// TIA Portal V18 export
// export: Created 2026-06-23T08:49:31.5753416Z, ExportSetting WithDefaults, DisplayName Totally Integrated Automation Portal, DisplayVersion V18, DisplayName TIA Portal Openness, DisplayVersion V18, DisplayName TIA Portal Version Control Interface, DisplayVersion V18, DisplayName STEP 7 Professional, DisplayVersion V18, DisplayName STEP 7 Safety, DisplayVersion V18, DisplayName WinCC Professional, DisplayVersion V18
FUNCTION "FC_Manual_Control_PLC2" : Void   // FC62, LAD
{ S7_Optimized_Access := 'TRUE' }
VERSION : 0.1
// stored: AutoNumber true, IsIECCheckEnabled false, SetENOAutomatically false, UDAEnableTagReadback false
BEGIN

REGION Network 1: Xác định trạng thái Manual Mode Active PLC2
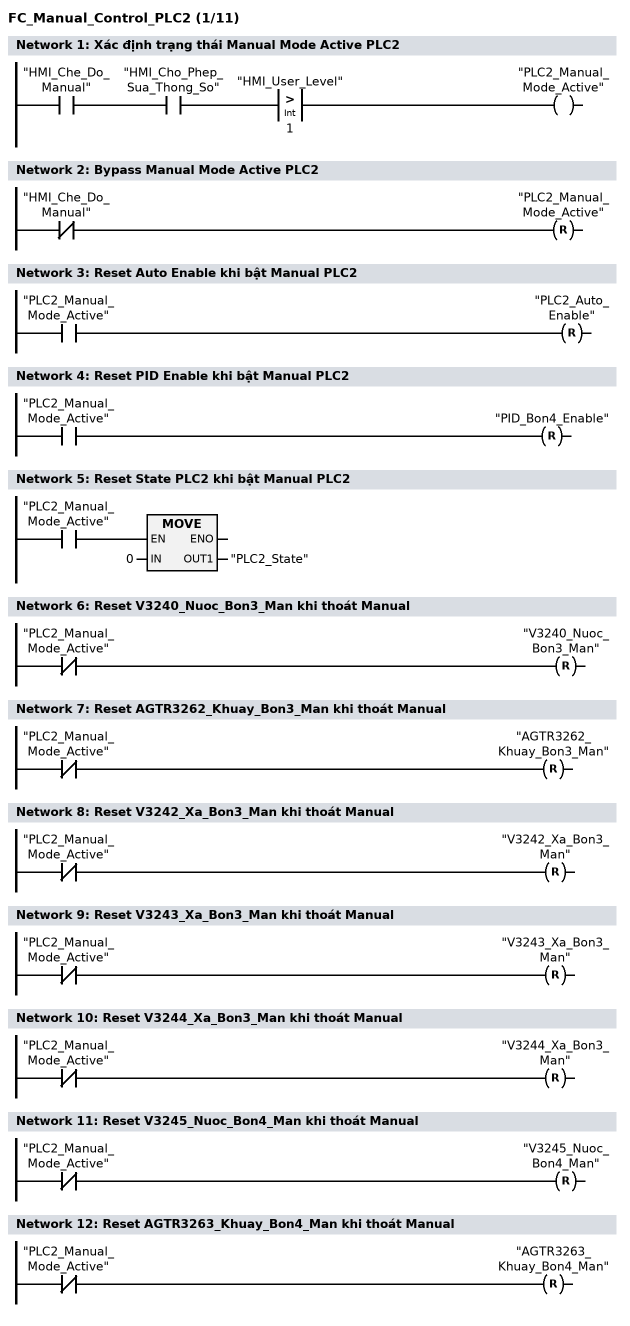
   RUNG wire#powerrail
      Contact( "HMI_Che_Do_Manual" )
      Contact( "HMI_Cho_Phep_Sua_Thong_So" )
      { S7_Templates := "SrcType := Int" } GT_Contact(in1 := "HMI_User_Level", in2 := 1)
      Coil( "PLC2_Manual_Mode_Active" )
   END_RUNG
   // the same network as SCL:
   "PLC2_Manual_Mode_Active" := "HMI_Che_Do_Manual" AND "HMI_Cho_Phep_Sua_Thong_So" AND ("HMI_User_Level" > 1);
END_REGION

REGION Network 2: Bypass Manual Mode Active PLC2
   RUNG wire#powerrail
      I_Contact( "HMI_Che_Do_Manual" )
      R_Coil( "PLC2_Manual_Mode_Active" )
   END_RUNG
   // the same network as SCL:
   IF NOT "HMI_Che_Do_Manual" THEN "PLC2_Manual_Mode_Active" := FALSE; END_IF;
END_REGION

REGION Network 3: Reset Auto Enable khi bật Manual PLC2
   RUNG wire#powerrail
      Contact( "PLC2_Manual_Mode_Active" )
      R_Coil( "PLC2_Auto_Enable" )
   END_RUNG
   // the same network as SCL:
   IF "PLC2_Manual_Mode_Active" THEN "PLC2_Auto_Enable" := FALSE; END_IF;
END_REGION

REGION Network 4: Reset PID Enable khi bật Manual PLC2
   RUNG wire#powerrail
      Contact( "PLC2_Manual_Mode_Active" )
      R_Coil( "PID_Bon4_Enable" )
   END_RUNG
   // the same network as SCL:
   IF "PLC2_Manual_Mode_Active" THEN "PID_Bon4_Enable" := FALSE; END_IF;
END_REGION

REGION Network 5: Reset State PLC2 khi bật Manual PLC2
   RUNG wire#powerrail
      Contact( "PLC2_Manual_Mode_Active" )
      { S7_GenerateENO := "TRUE" } Move(in := 0, out1 => "PLC2_State")
   END_RUNG
   // the same network as SCL:
   IF "PLC2_Manual_Mode_Active" THEN "PLC2_State" := 0; END_IF;
END_REGION

REGION Network 6: Reset V3240_Nuoc_Bon3_Man khi thoát Manual
   RUNG wire#powerrail
      I_Contact( "PLC2_Manual_Mode_Active" )
      R_Coil( "V3240_Nuoc_Bon3_Man" )
   END_RUNG
   // the same network as SCL:
   IF NOT "PLC2_Manual_Mode_Active" THEN "V3240_Nuoc_Bon3_Man" := FALSE; END_IF;
END_REGION

REGION Network 7: Reset AGTR3262_Khuay_Bon3_Man khi thoát Manual
   RUNG wire#powerrail
      I_Contact( "PLC2_Manual_Mode_Active" )
      R_Coil( "AGTR3262_Khuay_Bon3_Man" )
   END_RUNG
   // the same network as SCL:
   IF NOT "PLC2_Manual_Mode_Active" THEN "AGTR3262_Khuay_Bon3_Man" := FALSE; END_IF;
END_REGION

REGION Network 8: Reset V3242_Xa_Bon3_Man khi thoát Manual
   RUNG wire#powerrail
      I_Contact( "PLC2_Manual_Mode_Active" )
      R_Coil( "V3242_Xa_Bon3_Man" )
   END_RUNG
   // the same network as SCL:
   IF NOT "PLC2_Manual_Mode_Active" THEN "V3242_Xa_Bon3_Man" := FALSE; END_IF;
END_REGION

REGION Network 9: Reset V3243_Xa_Bon3_Man khi thoát Manual
   RUNG wire#powerrail
      I_Contact( "PLC2_Manual_Mode_Active" )
      R_Coil( "V3243_Xa_Bon3_Man" )
   END_RUNG
   // the same network as SCL:
   IF NOT "PLC2_Manual_Mode_Active" THEN "V3243_Xa_Bon3_Man" := FALSE; END_IF;
END_REGION

REGION Network 10: Reset V3244_Xa_Bon3_Man khi thoát Manual
   RUNG wire#powerrail
      I_Contact( "PLC2_Manual_Mode_Active" )
      R_Coil( "V3244_Xa_Bon3_Man" )
   END_RUNG
   // the same network as SCL:
   IF NOT "PLC2_Manual_Mode_Active" THEN "V3244_Xa_Bon3_Man" := FALSE; END_IF;
END_REGION

REGION Network 11: Reset V3245_Nuoc_Bon4_Man khi thoát Manual
   RUNG wire#powerrail
      I_Contact( "PLC2_Manual_Mode_Active" )
      R_Coil( "V3245_Nuoc_Bon4_Man" )
   END_RUNG
   // the same network as SCL:
   IF NOT "PLC2_Manual_Mode_Active" THEN "V3245_Nuoc_Bon4_Man" := FALSE; END_IF;
END_REGION

REGION Network 12: Reset AGTR3263_Khuay_Bon4_Man khi thoát Manual
   RUNG wire#powerrail
      I_Contact( "PLC2_Manual_Mode_Active" )
      R_Coil( "AGTR3263_Khuay_Bon4_Man" )
   END_RUNG
   // the same network as SCL:
   IF NOT "PLC2_Manual_Mode_Active" THEN "AGTR3263_Khuay_Bon4_Man" := FALSE; END_IF;
END_REGION

REGION Network 13: Reset AGTR3263_Dao_Chieu_Man khi thoát Manual
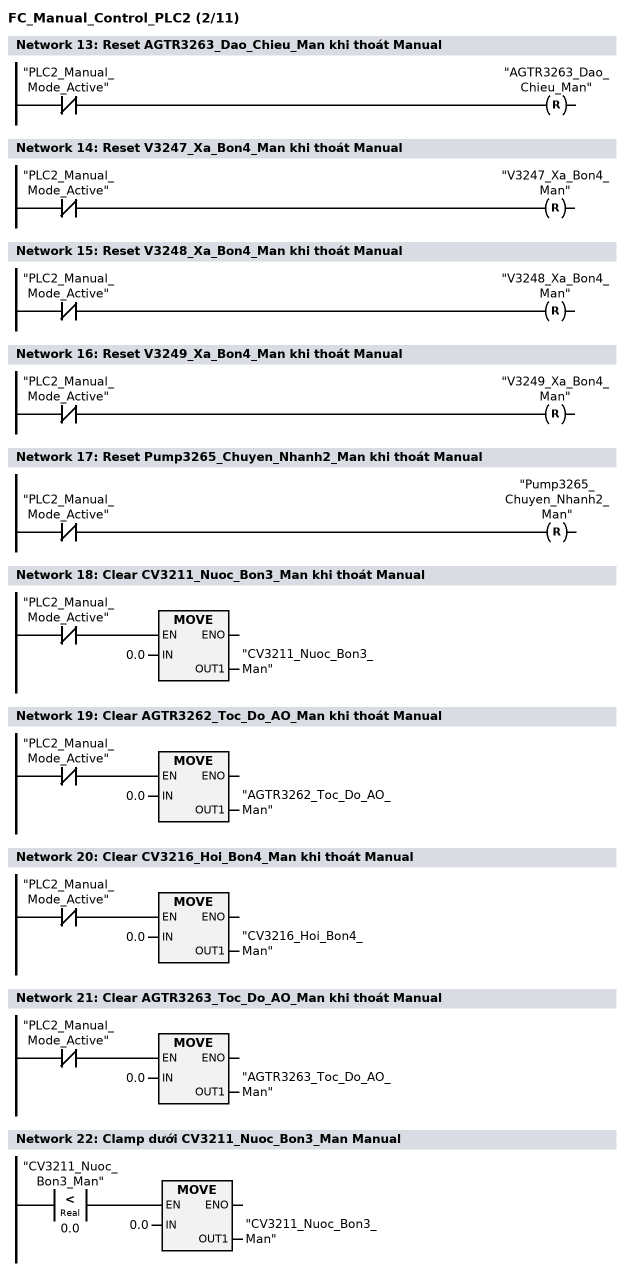
   RUNG wire#powerrail
      I_Contact( "PLC2_Manual_Mode_Active" )
      R_Coil( "AGTR3263_Dao_Chieu_Man" )
   END_RUNG
   // the same network as SCL:
   IF NOT "PLC2_Manual_Mode_Active" THEN "AGTR3263_Dao_Chieu_Man" := FALSE; END_IF;
END_REGION

REGION Network 14: Reset V3247_Xa_Bon4_Man khi thoát Manual
   RUNG wire#powerrail
      I_Contact( "PLC2_Manual_Mode_Active" )
      R_Coil( "V3247_Xa_Bon4_Man" )
   END_RUNG
   // the same network as SCL:
   IF NOT "PLC2_Manual_Mode_Active" THEN "V3247_Xa_Bon4_Man" := FALSE; END_IF;
END_REGION

REGION Network 15: Reset V3248_Xa_Bon4_Man khi thoát Manual
   RUNG wire#powerrail
      I_Contact( "PLC2_Manual_Mode_Active" )
      R_Coil( "V3248_Xa_Bon4_Man" )
   END_RUNG
   // the same network as SCL:
   IF NOT "PLC2_Manual_Mode_Active" THEN "V3248_Xa_Bon4_Man" := FALSE; END_IF;
END_REGION

REGION Network 16: Reset V3249_Xa_Bon4_Man khi thoát Manual
   RUNG wire#powerrail
      I_Contact( "PLC2_Manual_Mode_Active" )
      R_Coil( "V3249_Xa_Bon4_Man" )
   END_RUNG
   // the same network as SCL:
   IF NOT "PLC2_Manual_Mode_Active" THEN "V3249_Xa_Bon4_Man" := FALSE; END_IF;
END_REGION

REGION Network 17: Reset Pump3265_Chuyen_Nhanh2_Man khi thoát Manual
   RUNG wire#powerrail
      I_Contact( "PLC2_Manual_Mode_Active" )
      R_Coil( "Pump3265_Chuyen_Nhanh2_Man" )
   END_RUNG
   // the same network as SCL:
   IF NOT "PLC2_Manual_Mode_Active" THEN "Pump3265_Chuyen_Nhanh2_Man" := FALSE; END_IF;
END_REGION

REGION Network 18: Clear CV3211_Nuoc_Bon3_Man khi thoát Manual
   RUNG wire#powerrail
      I_Contact( "PLC2_Manual_Mode_Active" )
      { S7_GenerateENO := "TRUE" } Move(in := 0.0, out1 => "CV3211_Nuoc_Bon3_Man")
   END_RUNG
   // the same network as SCL:
   IF NOT "PLC2_Manual_Mode_Active" THEN "CV3211_Nuoc_Bon3_Man" := 0.0; END_IF;
END_REGION

REGION Network 19: Clear AGTR3262_Toc_Do_AO_Man khi thoát Manual
   RUNG wire#powerrail
      I_Contact( "PLC2_Manual_Mode_Active" )
      { S7_GenerateENO := "TRUE" } Move(in := 0.0, out1 => "AGTR3262_Toc_Do_AO_Man")
   END_RUNG
   // the same network as SCL:
   IF NOT "PLC2_Manual_Mode_Active" THEN "AGTR3262_Toc_Do_AO_Man" := 0.0; END_IF;
END_REGION

REGION Network 20: Clear CV3216_Hoi_Bon4_Man khi thoát Manual
   RUNG wire#powerrail
      I_Contact( "PLC2_Manual_Mode_Active" )
      { S7_GenerateENO := "TRUE" } Move(in := 0.0, out1 => "CV3216_Hoi_Bon4_Man")
   END_RUNG
   // the same network as SCL:
   IF NOT "PLC2_Manual_Mode_Active" THEN "CV3216_Hoi_Bon4_Man" := 0.0; END_IF;
END_REGION

REGION Network 21: Clear AGTR3263_Toc_Do_AO_Man khi thoát Manual
   RUNG wire#powerrail
      I_Contact( "PLC2_Manual_Mode_Active" )
      { S7_GenerateENO := "TRUE" } Move(in := 0.0, out1 => "AGTR3263_Toc_Do_AO_Man")
   END_RUNG
   // the same network as SCL:
   IF NOT "PLC2_Manual_Mode_Active" THEN "AGTR3263_Toc_Do_AO_Man" := 0.0; END_IF;
END_REGION

REGION Network 22: Clamp dưới CV3211_Nuoc_Bon3_Man Manual
   RUNG wire#powerrail
      { S7_Templates := "SrcType := Real" } LT_Contact(in1 := "CV3211_Nuoc_Bon3_Man", in2 := 0.0)
      { S7_GenerateENO := "TRUE" } Move(in := 0.0, out1 => "CV3211_Nuoc_Bon3_Man")
   END_RUNG
   // the same network as SCL:
   IF "CV3211_Nuoc_Bon3_Man" < 0.0 THEN "CV3211_Nuoc_Bon3_Man" := 0.0; END_IF;
END_REGION

REGION Network 23: Clamp trên CV3211_Nuoc_Bon3_Man Manual
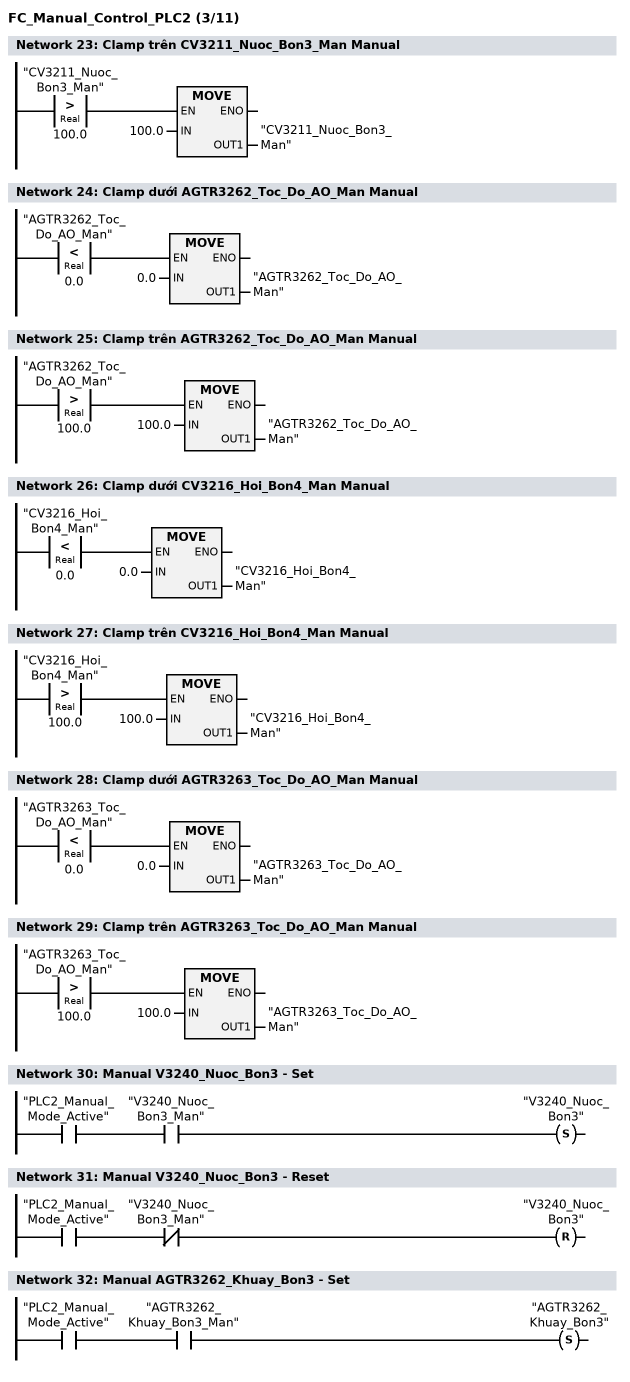
   RUNG wire#powerrail
      { S7_Templates := "SrcType := Real" } GT_Contact(in1 := "CV3211_Nuoc_Bon3_Man", in2 := 100.0)
      { S7_GenerateENO := "TRUE" } Move(in := 100.0, out1 => "CV3211_Nuoc_Bon3_Man")
   END_RUNG
   // the same network as SCL:
   IF "CV3211_Nuoc_Bon3_Man" > 100.0 THEN "CV3211_Nuoc_Bon3_Man" := 100.0; END_IF;
END_REGION

REGION Network 24: Clamp dưới AGTR3262_Toc_Do_AO_Man Manual
   RUNG wire#powerrail
      { S7_Templates := "SrcType := Real" } LT_Contact(in1 := "AGTR3262_Toc_Do_AO_Man", in2 := 0.0)
      { S7_GenerateENO := "TRUE" } Move(in := 0.0, out1 => "AGTR3262_Toc_Do_AO_Man")
   END_RUNG
   // the same network as SCL:
   IF "AGTR3262_Toc_Do_AO_Man" < 0.0 THEN "AGTR3262_Toc_Do_AO_Man" := 0.0; END_IF;
END_REGION

REGION Network 25: Clamp trên AGTR3262_Toc_Do_AO_Man Manual
   RUNG wire#powerrail
      { S7_Templates := "SrcType := Real" } GT_Contact(in1 := "AGTR3262_Toc_Do_AO_Man", in2 := 100.0)
      { S7_GenerateENO := "TRUE" } Move(in := 100.0, out1 => "AGTR3262_Toc_Do_AO_Man")
   END_RUNG
   // the same network as SCL:
   IF "AGTR3262_Toc_Do_AO_Man" > 100.0 THEN "AGTR3262_Toc_Do_AO_Man" := 100.0; END_IF;
END_REGION

REGION Network 26: Clamp dưới CV3216_Hoi_Bon4_Man Manual
   RUNG wire#powerrail
      { S7_Templates := "SrcType := Real" } LT_Contact(in1 := "CV3216_Hoi_Bon4_Man", in2 := 0.0)
      { S7_GenerateENO := "TRUE" } Move(in := 0.0, out1 => "CV3216_Hoi_Bon4_Man")
   END_RUNG
   // the same network as SCL:
   IF "CV3216_Hoi_Bon4_Man" < 0.0 THEN "CV3216_Hoi_Bon4_Man" := 0.0; END_IF;
END_REGION

REGION Network 27: Clamp trên CV3216_Hoi_Bon4_Man Manual
   RUNG wire#powerrail
      { S7_Templates := "SrcType := Real" } GT_Contact(in1 := "CV3216_Hoi_Bon4_Man", in2 := 100.0)
      { S7_GenerateENO := "TRUE" } Move(in := 100.0, out1 => "CV3216_Hoi_Bon4_Man")
   END_RUNG
   // the same network as SCL:
   IF "CV3216_Hoi_Bon4_Man" > 100.0 THEN "CV3216_Hoi_Bon4_Man" := 100.0; END_IF;
END_REGION

REGION Network 28: Clamp dưới AGTR3263_Toc_Do_AO_Man Manual
   RUNG wire#powerrail
      { S7_Templates := "SrcType := Real" } LT_Contact(in1 := "AGTR3263_Toc_Do_AO_Man", in2 := 0.0)
      { S7_GenerateENO := "TRUE" } Move(in := 0.0, out1 => "AGTR3263_Toc_Do_AO_Man")
   END_RUNG
   // the same network as SCL:
   IF "AGTR3263_Toc_Do_AO_Man" < 0.0 THEN "AGTR3263_Toc_Do_AO_Man" := 0.0; END_IF;
END_REGION

REGION Network 29: Clamp trên AGTR3263_Toc_Do_AO_Man Manual
   RUNG wire#powerrail
      { S7_Templates := "SrcType := Real" } GT_Contact(in1 := "AGTR3263_Toc_Do_AO_Man", in2 := 100.0)
      { S7_GenerateENO := "TRUE" } Move(in := 100.0, out1 => "AGTR3263_Toc_Do_AO_Man")
   END_RUNG
   // the same network as SCL:
   IF "AGTR3263_Toc_Do_AO_Man" > 100.0 THEN "AGTR3263_Toc_Do_AO_Man" := 100.0; END_IF;
END_REGION

REGION Network 30: Manual V3240_Nuoc_Bon3 - Set
   RUNG wire#powerrail
      Contact( "PLC2_Manual_Mode_Active" )
      Contact( "V3240_Nuoc_Bon3_Man" )
      S_Coil( "V3240_Nuoc_Bon3" )
   END_RUNG
   // the same network as SCL:
   IF "PLC2_Manual_Mode_Active" AND "V3240_Nuoc_Bon3_Man" THEN "V3240_Nuoc_Bon3" := TRUE; END_IF;
END_REGION

REGION Network 31: Manual V3240_Nuoc_Bon3 - Reset
   RUNG wire#powerrail
      Contact( "PLC2_Manual_Mode_Active" )
      I_Contact( "V3240_Nuoc_Bon3_Man" )
      R_Coil( "V3240_Nuoc_Bon3" )
   END_RUNG
   // the same network as SCL:
   IF "PLC2_Manual_Mode_Active" AND NOT "V3240_Nuoc_Bon3_Man" THEN "V3240_Nuoc_Bon3" := FALSE; END_IF;
END_REGION

REGION Network 32: Manual AGTR3262_Khuay_Bon3 - Set
   RUNG wire#powerrail
      Contact( "PLC2_Manual_Mode_Active" )
      Contact( "AGTR3262_Khuay_Bon3_Man" )
      S_Coil( "AGTR3262_Khuay_Bon3" )
   END_RUNG
   // the same network as SCL:
   IF "PLC2_Manual_Mode_Active" AND "AGTR3262_Khuay_Bon3_Man" THEN "AGTR3262_Khuay_Bon3" := TRUE; END_IF;
END_REGION

REGION Network 33: Manual AGTR3262_Khuay_Bon3 - Reset
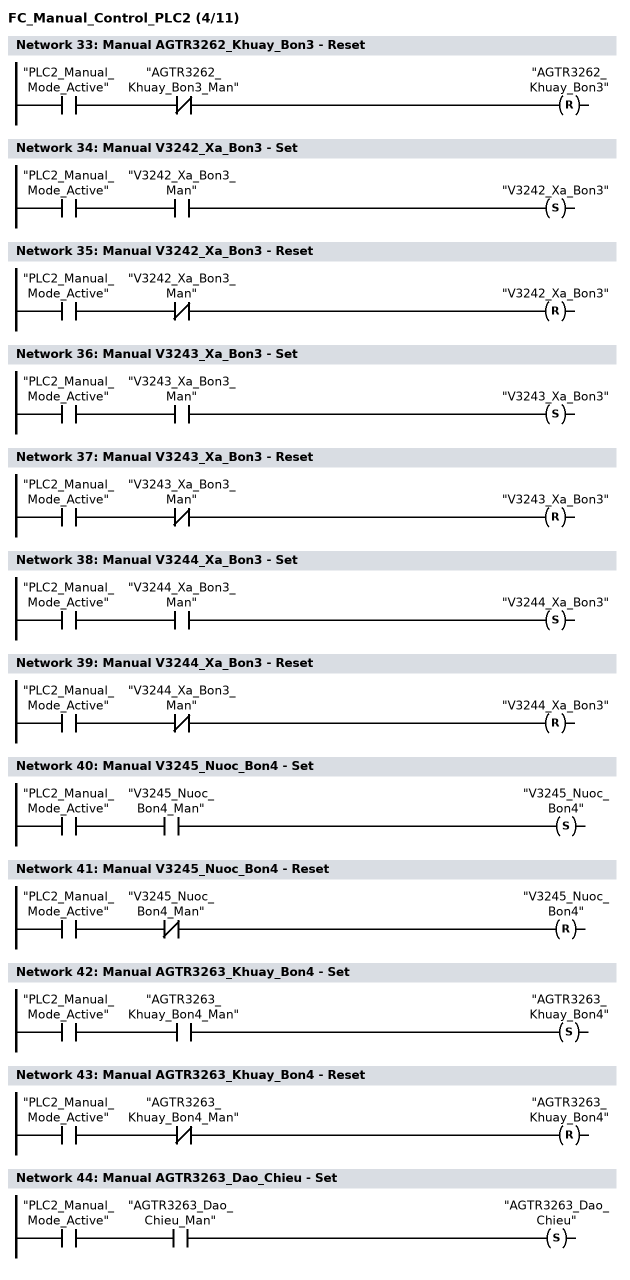
   RUNG wire#powerrail
      Contact( "PLC2_Manual_Mode_Active" )
      I_Contact( "AGTR3262_Khuay_Bon3_Man" )
      R_Coil( "AGTR3262_Khuay_Bon3" )
   END_RUNG
   // the same network as SCL:
   IF "PLC2_Manual_Mode_Active" AND NOT "AGTR3262_Khuay_Bon3_Man" THEN
       "AGTR3262_Khuay_Bon3" := FALSE;
   END_IF;
END_REGION

REGION Network 34: Manual V3242_Xa_Bon3 - Set
   RUNG wire#powerrail
      Contact( "PLC2_Manual_Mode_Active" )
      Contact( "V3242_Xa_Bon3_Man" )
      S_Coil( "V3242_Xa_Bon3" )
   END_RUNG
   // the same network as SCL:
   IF "PLC2_Manual_Mode_Active" AND "V3242_Xa_Bon3_Man" THEN "V3242_Xa_Bon3" := TRUE; END_IF;
END_REGION

REGION Network 35: Manual V3242_Xa_Bon3 - Reset
   RUNG wire#powerrail
      Contact( "PLC2_Manual_Mode_Active" )
      I_Contact( "V3242_Xa_Bon3_Man" )
      R_Coil( "V3242_Xa_Bon3" )
   END_RUNG
   // the same network as SCL:
   IF "PLC2_Manual_Mode_Active" AND NOT "V3242_Xa_Bon3_Man" THEN "V3242_Xa_Bon3" := FALSE; END_IF;
END_REGION

REGION Network 36: Manual V3243_Xa_Bon3 - Set
   RUNG wire#powerrail
      Contact( "PLC2_Manual_Mode_Active" )
      Contact( "V3243_Xa_Bon3_Man" )
      S_Coil( "V3243_Xa_Bon3" )
   END_RUNG
   // the same network as SCL:
   IF "PLC2_Manual_Mode_Active" AND "V3243_Xa_Bon3_Man" THEN "V3243_Xa_Bon3" := TRUE; END_IF;
END_REGION

REGION Network 37: Manual V3243_Xa_Bon3 - Reset
   RUNG wire#powerrail
      Contact( "PLC2_Manual_Mode_Active" )
      I_Contact( "V3243_Xa_Bon3_Man" )
      R_Coil( "V3243_Xa_Bon3" )
   END_RUNG
   // the same network as SCL:
   IF "PLC2_Manual_Mode_Active" AND NOT "V3243_Xa_Bon3_Man" THEN "V3243_Xa_Bon3" := FALSE; END_IF;
END_REGION

REGION Network 38: Manual V3244_Xa_Bon3 - Set
   RUNG wire#powerrail
      Contact( "PLC2_Manual_Mode_Active" )
      Contact( "V3244_Xa_Bon3_Man" )
      S_Coil( "V3244_Xa_Bon3" )
   END_RUNG
   // the same network as SCL:
   IF "PLC2_Manual_Mode_Active" AND "V3244_Xa_Bon3_Man" THEN "V3244_Xa_Bon3" := TRUE; END_IF;
END_REGION

REGION Network 39: Manual V3244_Xa_Bon3 - Reset
   RUNG wire#powerrail
      Contact( "PLC2_Manual_Mode_Active" )
      I_Contact( "V3244_Xa_Bon3_Man" )
      R_Coil( "V3244_Xa_Bon3" )
   END_RUNG
   // the same network as SCL:
   IF "PLC2_Manual_Mode_Active" AND NOT "V3244_Xa_Bon3_Man" THEN "V3244_Xa_Bon3" := FALSE; END_IF;
END_REGION

REGION Network 40: Manual V3245_Nuoc_Bon4 - Set
   RUNG wire#powerrail
      Contact( "PLC2_Manual_Mode_Active" )
      Contact( "V3245_Nuoc_Bon4_Man" )
      S_Coil( "V3245_Nuoc_Bon4" )
   END_RUNG
   // the same network as SCL:
   IF "PLC2_Manual_Mode_Active" AND "V3245_Nuoc_Bon4_Man" THEN "V3245_Nuoc_Bon4" := TRUE; END_IF;
END_REGION

REGION Network 41: Manual V3245_Nuoc_Bon4 - Reset
   RUNG wire#powerrail
      Contact( "PLC2_Manual_Mode_Active" )
      I_Contact( "V3245_Nuoc_Bon4_Man" )
      R_Coil( "V3245_Nuoc_Bon4" )
   END_RUNG
   // the same network as SCL:
   IF "PLC2_Manual_Mode_Active" AND NOT "V3245_Nuoc_Bon4_Man" THEN "V3245_Nuoc_Bon4" := FALSE; END_IF;
END_REGION

REGION Network 42: Manual AGTR3263_Khuay_Bon4 - Set
   RUNG wire#powerrail
      Contact( "PLC2_Manual_Mode_Active" )
      Contact( "AGTR3263_Khuay_Bon4_Man" )
      S_Coil( "AGTR3263_Khuay_Bon4" )
   END_RUNG
   // the same network as SCL:
   IF "PLC2_Manual_Mode_Active" AND "AGTR3263_Khuay_Bon4_Man" THEN "AGTR3263_Khuay_Bon4" := TRUE; END_IF;
END_REGION

REGION Network 43: Manual AGTR3263_Khuay_Bon4 - Reset
   RUNG wire#powerrail
      Contact( "PLC2_Manual_Mode_Active" )
      I_Contact( "AGTR3263_Khuay_Bon4_Man" )
      R_Coil( "AGTR3263_Khuay_Bon4" )
   END_RUNG
   // the same network as SCL:
   IF "PLC2_Manual_Mode_Active" AND NOT "AGTR3263_Khuay_Bon4_Man" THEN
       "AGTR3263_Khuay_Bon4" := FALSE;
   END_IF;
END_REGION

REGION Network 44: Manual AGTR3263_Dao_Chieu - Set
   RUNG wire#powerrail
      Contact( "PLC2_Manual_Mode_Active" )
      Contact( "AGTR3263_Dao_Chieu_Man" )
      S_Coil( "AGTR3263_Dao_Chieu" )
   END_RUNG
   // the same network as SCL:
   IF "PLC2_Manual_Mode_Active" AND "AGTR3263_Dao_Chieu_Man" THEN "AGTR3263_Dao_Chieu" := TRUE; END_IF;
END_REGION

REGION Network 45: Manual AGTR3263_Dao_Chieu - Reset
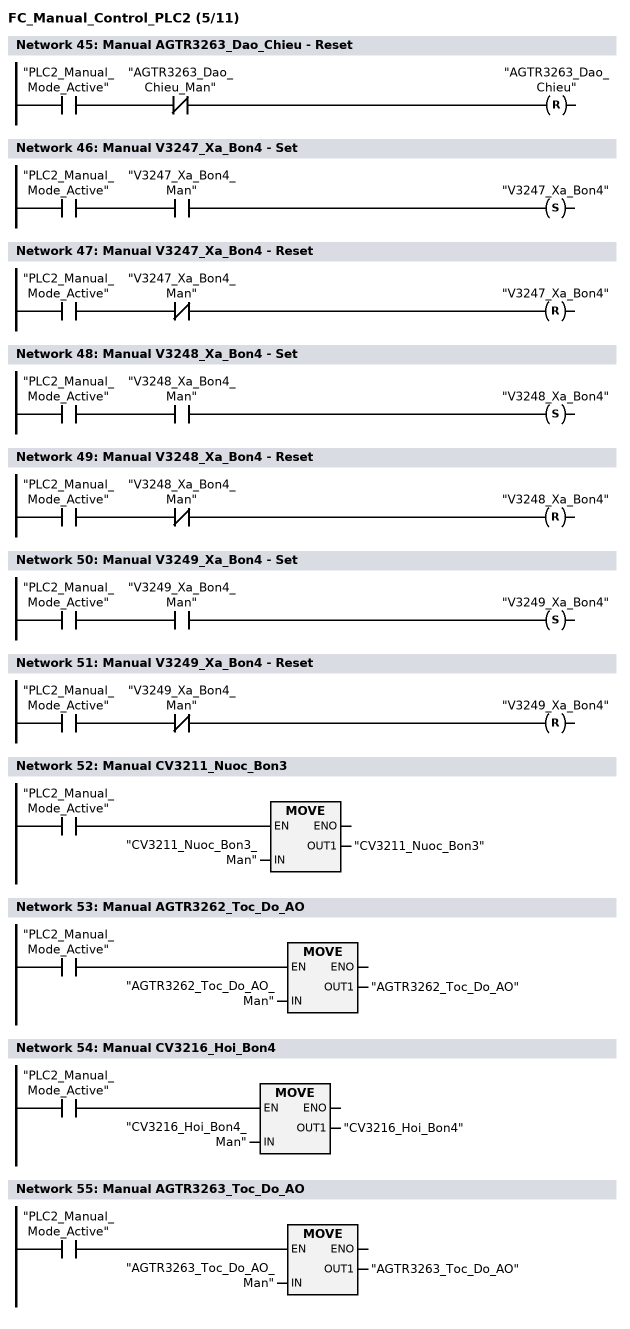
   RUNG wire#powerrail
      Contact( "PLC2_Manual_Mode_Active" )
      I_Contact( "AGTR3263_Dao_Chieu_Man" )
      R_Coil( "AGTR3263_Dao_Chieu" )
   END_RUNG
   // the same network as SCL:
   IF "PLC2_Manual_Mode_Active" AND NOT "AGTR3263_Dao_Chieu_Man" THEN "AGTR3263_Dao_Chieu" := FALSE; END_IF;
END_REGION

REGION Network 46: Manual V3247_Xa_Bon4 - Set
   RUNG wire#powerrail
      Contact( "PLC2_Manual_Mode_Active" )
      Contact( "V3247_Xa_Bon4_Man" )
      S_Coil( "V3247_Xa_Bon4" )
   END_RUNG
   // the same network as SCL:
   IF "PLC2_Manual_Mode_Active" AND "V3247_Xa_Bon4_Man" THEN "V3247_Xa_Bon4" := TRUE; END_IF;
END_REGION

REGION Network 47: Manual V3247_Xa_Bon4 - Reset
   RUNG wire#powerrail
      Contact( "PLC2_Manual_Mode_Active" )
      I_Contact( "V3247_Xa_Bon4_Man" )
      R_Coil( "V3247_Xa_Bon4" )
   END_RUNG
   // the same network as SCL:
   IF "PLC2_Manual_Mode_Active" AND NOT "V3247_Xa_Bon4_Man" THEN "V3247_Xa_Bon4" := FALSE; END_IF;
END_REGION

REGION Network 48: Manual V3248_Xa_Bon4 - Set
   RUNG wire#powerrail
      Contact( "PLC2_Manual_Mode_Active" )
      Contact( "V3248_Xa_Bon4_Man" )
      S_Coil( "V3248_Xa_Bon4" )
   END_RUNG
   // the same network as SCL:
   IF "PLC2_Manual_Mode_Active" AND "V3248_Xa_Bon4_Man" THEN "V3248_Xa_Bon4" := TRUE; END_IF;
END_REGION

REGION Network 49: Manual V3248_Xa_Bon4 - Reset
   RUNG wire#powerrail
      Contact( "PLC2_Manual_Mode_Active" )
      I_Contact( "V3248_Xa_Bon4_Man" )
      R_Coil( "V3248_Xa_Bon4" )
   END_RUNG
   // the same network as SCL:
   IF "PLC2_Manual_Mode_Active" AND NOT "V3248_Xa_Bon4_Man" THEN "V3248_Xa_Bon4" := FALSE; END_IF;
END_REGION

REGION Network 50: Manual V3249_Xa_Bon4 - Set
   RUNG wire#powerrail
      Contact( "PLC2_Manual_Mode_Active" )
      Contact( "V3249_Xa_Bon4_Man" )
      S_Coil( "V3249_Xa_Bon4" )
   END_RUNG
   // the same network as SCL:
   IF "PLC2_Manual_Mode_Active" AND "V3249_Xa_Bon4_Man" THEN "V3249_Xa_Bon4" := TRUE; END_IF;
END_REGION

REGION Network 51: Manual V3249_Xa_Bon4 - Reset
   RUNG wire#powerrail
      Contact( "PLC2_Manual_Mode_Active" )
      I_Contact( "V3249_Xa_Bon4_Man" )
      R_Coil( "V3249_Xa_Bon4" )
   END_RUNG
   // the same network as SCL:
   IF "PLC2_Manual_Mode_Active" AND NOT "V3249_Xa_Bon4_Man" THEN "V3249_Xa_Bon4" := FALSE; END_IF;
END_REGION

REGION Network 52: Manual CV3211_Nuoc_Bon3
   RUNG wire#powerrail
      Contact( "PLC2_Manual_Mode_Active" )
      { S7_GenerateENO := "TRUE" } Move(in := "CV3211_Nuoc_Bon3_Man", out1 => "CV3211_Nuoc_Bon3")
   END_RUNG
   // the same network as SCL:
   IF "PLC2_Manual_Mode_Active" THEN "CV3211_Nuoc_Bon3" := "CV3211_Nuoc_Bon3_Man"; END_IF;
END_REGION

REGION Network 53: Manual AGTR3262_Toc_Do_AO
   RUNG wire#powerrail
      Contact( "PLC2_Manual_Mode_Active" )
      { S7_GenerateENO := "TRUE" } Move(in := "AGTR3262_Toc_Do_AO_Man", out1 => "AGTR3262_Toc_Do_AO")
   END_RUNG
   // the same network as SCL:
   IF "PLC2_Manual_Mode_Active" THEN "AGTR3262_Toc_Do_AO" := "AGTR3262_Toc_Do_AO_Man"; END_IF;
END_REGION

REGION Network 54: Manual CV3216_Hoi_Bon4
   RUNG wire#powerrail
      Contact( "PLC2_Manual_Mode_Active" )
      { S7_GenerateENO := "TRUE" } Move(in := "CV3216_Hoi_Bon4_Man", out1 => "CV3216_Hoi_Bon4")
   END_RUNG
   // the same network as SCL:
   IF "PLC2_Manual_Mode_Active" THEN "CV3216_Hoi_Bon4" := "CV3216_Hoi_Bon4_Man"; END_IF;
END_REGION

REGION Network 55: Manual AGTR3263_Toc_Do_AO
   RUNG wire#powerrail
      Contact( "PLC2_Manual_Mode_Active" )
      { S7_GenerateENO := "TRUE" } Move(in := "AGTR3263_Toc_Do_AO_Man", out1 => "AGTR3263_Toc_Do_AO")
   END_RUNG
   // the same network as SCL:
   IF "PLC2_Manual_Mode_Active" THEN "AGTR3263_Toc_Do_AO" := "AGTR3263_Toc_Do_AO_Man"; END_IF;
END_REGION

REGION Network 56: Manual Pump3265_Chuyen_Nhanh2 - Safe Reset
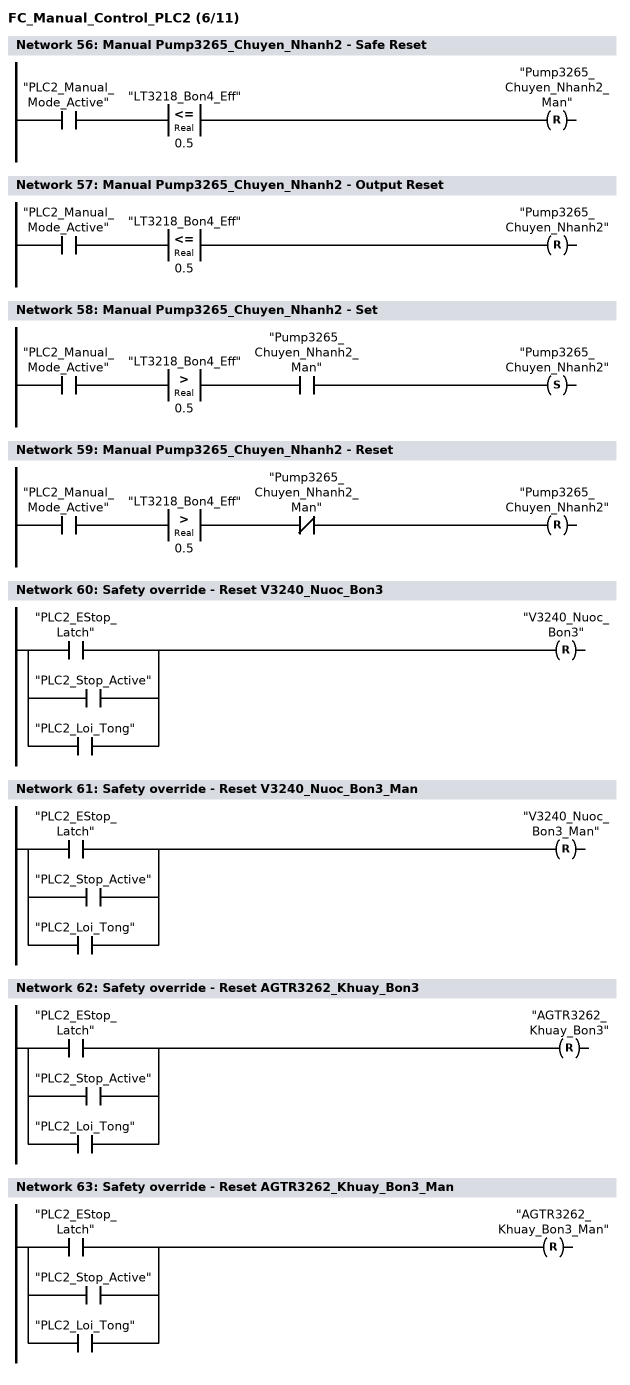
   RUNG wire#powerrail
      Contact( "PLC2_Manual_Mode_Active" )
      { S7_Templates := "SrcType := Real" } LE_Contact(in1 := "LT3218_Bon4_Eff", in2 := 0.5)
      R_Coil( "Pump3265_Chuyen_Nhanh2_Man" )
   END_RUNG
   // the same network as SCL:
   IF "PLC2_Manual_Mode_Active" AND ("LT3218_Bon4_Eff" <= 0.5) THEN
       "Pump3265_Chuyen_Nhanh2_Man" := FALSE;
   END_IF;
END_REGION

REGION Network 57: Manual Pump3265_Chuyen_Nhanh2 - Output Reset
   RUNG wire#powerrail
      Contact( "PLC2_Manual_Mode_Active" )
      { S7_Templates := "SrcType := Real" } LE_Contact(in1 := "LT3218_Bon4_Eff", in2 := 0.5)
      R_Coil( "Pump3265_Chuyen_Nhanh2" )
   END_RUNG
   // the same network as SCL:
   IF "PLC2_Manual_Mode_Active" AND ("LT3218_Bon4_Eff" <= 0.5) THEN
       "Pump3265_Chuyen_Nhanh2" := FALSE;
   END_IF;
END_REGION

REGION Network 58: Manual Pump3265_Chuyen_Nhanh2 - Set
   RUNG wire#powerrail
      Contact( "PLC2_Manual_Mode_Active" )
      { S7_Templates := "SrcType := Real" } GT_Contact(in1 := "LT3218_Bon4_Eff", in2 := 0.5)
      Contact( "Pump3265_Chuyen_Nhanh2_Man" )
      S_Coil( "Pump3265_Chuyen_Nhanh2" )
   END_RUNG
   // the same network as SCL:
   IF "PLC2_Manual_Mode_Active" AND ("LT3218_Bon4_Eff" > 0.5) AND "Pump3265_Chuyen_Nhanh2_Man" THEN
       "Pump3265_Chuyen_Nhanh2" := TRUE;
   END_IF;
END_REGION

REGION Network 59: Manual Pump3265_Chuyen_Nhanh2 - Reset
   RUNG wire#powerrail
      Contact( "PLC2_Manual_Mode_Active" )
      { S7_Templates := "SrcType := Real" } GT_Contact(in1 := "LT3218_Bon4_Eff", in2 := 0.5)
      I_Contact( "Pump3265_Chuyen_Nhanh2_Man" )
      R_Coil( "Pump3265_Chuyen_Nhanh2" )
   END_RUNG
   // the same network as SCL:
   IF "PLC2_Manual_Mode_Active" AND ("LT3218_Bon4_Eff" > 0.5) AND NOT "Pump3265_Chuyen_Nhanh2_Man" THEN
       "Pump3265_Chuyen_Nhanh2" := FALSE;
   END_IF;
END_REGION

REGION Network 60: Safety override - Reset V3240_Nuoc_Bon3
   RUNG wire#powerrail
      Contact( "PLC2_EStop_Latch" )
      wire#w1
      R_Coil( "V3240_Nuoc_Bon3" )
   END_RUNG
   RUNG wire#powerrail
      Contact( "PLC2_Stop_Active" )
   END_RUNG wire#w1
   RUNG wire#powerrail
      Contact( "PLC2_Loi_Tong" )
   END_RUNG wire#w1
   // the same network as SCL:
   IF "PLC2_EStop_Latch" OR "PLC2_Stop_Active" OR "PLC2_Loi_Tong" THEN "V3240_Nuoc_Bon3" := FALSE; END_IF;
END_REGION

REGION Network 61: Safety override - Reset V3240_Nuoc_Bon3_Man
   RUNG wire#powerrail
      Contact( "PLC2_EStop_Latch" )
      wire#w1
      R_Coil( "V3240_Nuoc_Bon3_Man" )
   END_RUNG
   RUNG wire#powerrail
      Contact( "PLC2_Stop_Active" )
   END_RUNG wire#w1
   RUNG wire#powerrail
      Contact( "PLC2_Loi_Tong" )
   END_RUNG wire#w1
   // the same network as SCL:
   IF "PLC2_EStop_Latch" OR "PLC2_Stop_Active" OR "PLC2_Loi_Tong" THEN
       "V3240_Nuoc_Bon3_Man" := FALSE;
   END_IF;
END_REGION

REGION Network 62: Safety override - Reset AGTR3262_Khuay_Bon3
   RUNG wire#powerrail
      Contact( "PLC2_EStop_Latch" )
      wire#w1
      R_Coil( "AGTR3262_Khuay_Bon3" )
   END_RUNG
   RUNG wire#powerrail
      Contact( "PLC2_Stop_Active" )
   END_RUNG wire#w1
   RUNG wire#powerrail
      Contact( "PLC2_Loi_Tong" )
   END_RUNG wire#w1
   // the same network as SCL:
   IF "PLC2_EStop_Latch" OR "PLC2_Stop_Active" OR "PLC2_Loi_Tong" THEN
       "AGTR3262_Khuay_Bon3" := FALSE;
   END_IF;
END_REGION

REGION Network 63: Safety override - Reset AGTR3262_Khuay_Bon3_Man
   RUNG wire#powerrail
      Contact( "PLC2_EStop_Latch" )
      wire#w1
      R_Coil( "AGTR3262_Khuay_Bon3_Man" )
   END_RUNG
   RUNG wire#powerrail
      Contact( "PLC2_Stop_Active" )
   END_RUNG wire#w1
   RUNG wire#powerrail
      Contact( "PLC2_Loi_Tong" )
   END_RUNG wire#w1
   // the same network as SCL:
   IF "PLC2_EStop_Latch" OR "PLC2_Stop_Active" OR "PLC2_Loi_Tong" THEN
       "AGTR3262_Khuay_Bon3_Man" := FALSE;
   END_IF;
END_REGION

REGION Network 64: Safety override - Reset V3242_Xa_Bon3
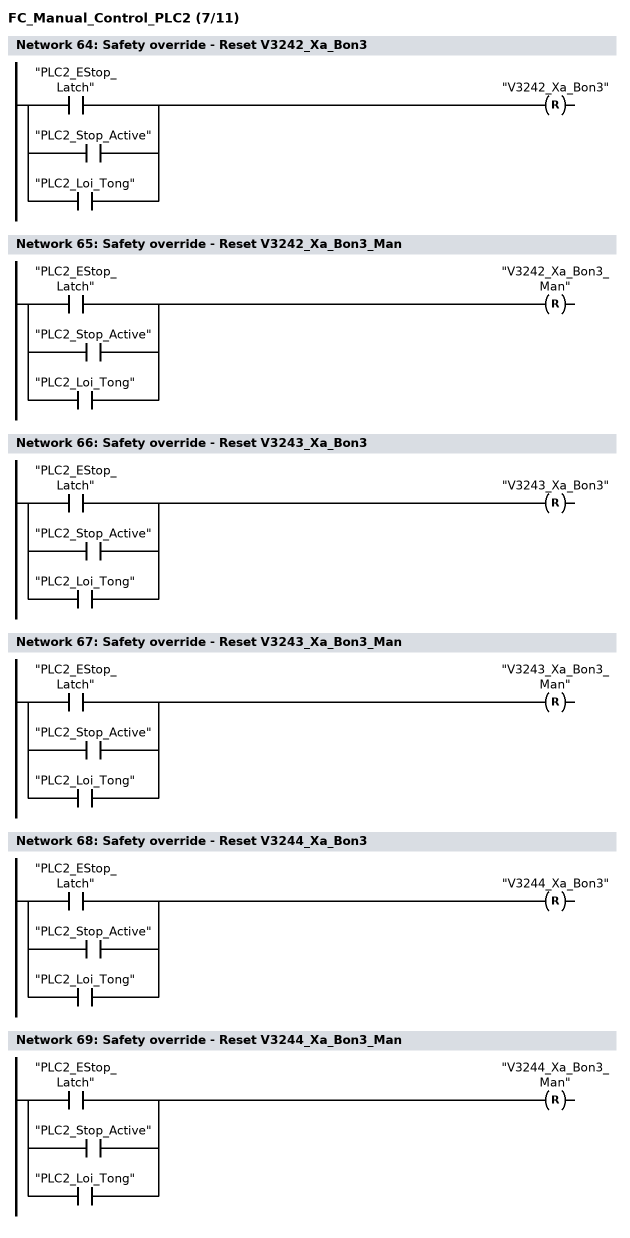
   RUNG wire#powerrail
      Contact( "PLC2_EStop_Latch" )
      wire#w1
      R_Coil( "V3242_Xa_Bon3" )
   END_RUNG
   RUNG wire#powerrail
      Contact( "PLC2_Stop_Active" )
   END_RUNG wire#w1
   RUNG wire#powerrail
      Contact( "PLC2_Loi_Tong" )
   END_RUNG wire#w1
   // the same network as SCL:
   IF "PLC2_EStop_Latch" OR "PLC2_Stop_Active" OR "PLC2_Loi_Tong" THEN "V3242_Xa_Bon3" := FALSE; END_IF;
END_REGION

REGION Network 65: Safety override - Reset V3242_Xa_Bon3_Man
   RUNG wire#powerrail
      Contact( "PLC2_EStop_Latch" )
      wire#w1
      R_Coil( "V3242_Xa_Bon3_Man" )
   END_RUNG
   RUNG wire#powerrail
      Contact( "PLC2_Stop_Active" )
   END_RUNG wire#w1
   RUNG wire#powerrail
      Contact( "PLC2_Loi_Tong" )
   END_RUNG wire#w1
   // the same network as SCL:
   IF "PLC2_EStop_Latch" OR "PLC2_Stop_Active" OR "PLC2_Loi_Tong" THEN "V3242_Xa_Bon3_Man" := FALSE; END_IF;
END_REGION

REGION Network 66: Safety override - Reset V3243_Xa_Bon3
   RUNG wire#powerrail
      Contact( "PLC2_EStop_Latch" )
      wire#w1
      R_Coil( "V3243_Xa_Bon3" )
   END_RUNG
   RUNG wire#powerrail
      Contact( "PLC2_Stop_Active" )
   END_RUNG wire#w1
   RUNG wire#powerrail
      Contact( "PLC2_Loi_Tong" )
   END_RUNG wire#w1
   // the same network as SCL:
   IF "PLC2_EStop_Latch" OR "PLC2_Stop_Active" OR "PLC2_Loi_Tong" THEN "V3243_Xa_Bon3" := FALSE; END_IF;
END_REGION

REGION Network 67: Safety override - Reset V3243_Xa_Bon3_Man
   RUNG wire#powerrail
      Contact( "PLC2_EStop_Latch" )
      wire#w1
      R_Coil( "V3243_Xa_Bon3_Man" )
   END_RUNG
   RUNG wire#powerrail
      Contact( "PLC2_Stop_Active" )
   END_RUNG wire#w1
   RUNG wire#powerrail
      Contact( "PLC2_Loi_Tong" )
   END_RUNG wire#w1
   // the same network as SCL:
   IF "PLC2_EStop_Latch" OR "PLC2_Stop_Active" OR "PLC2_Loi_Tong" THEN "V3243_Xa_Bon3_Man" := FALSE; END_IF;
END_REGION

REGION Network 68: Safety override - Reset V3244_Xa_Bon3
   RUNG wire#powerrail
      Contact( "PLC2_EStop_Latch" )
      wire#w1
      R_Coil( "V3244_Xa_Bon3" )
   END_RUNG
   RUNG wire#powerrail
      Contact( "PLC2_Stop_Active" )
   END_RUNG wire#w1
   RUNG wire#powerrail
      Contact( "PLC2_Loi_Tong" )
   END_RUNG wire#w1
   // the same network as SCL:
   IF "PLC2_EStop_Latch" OR "PLC2_Stop_Active" OR "PLC2_Loi_Tong" THEN "V3244_Xa_Bon3" := FALSE; END_IF;
END_REGION

REGION Network 69: Safety override - Reset V3244_Xa_Bon3_Man
   RUNG wire#powerrail
      Contact( "PLC2_EStop_Latch" )
      wire#w1
      R_Coil( "V3244_Xa_Bon3_Man" )
   END_RUNG
   RUNG wire#powerrail
      Contact( "PLC2_Stop_Active" )
   END_RUNG wire#w1
   RUNG wire#powerrail
      Contact( "PLC2_Loi_Tong" )
   END_RUNG wire#w1
   // the same network as SCL:
   IF "PLC2_EStop_Latch" OR "PLC2_Stop_Active" OR "PLC2_Loi_Tong" THEN "V3244_Xa_Bon3_Man" := FALSE; END_IF;
END_REGION

REGION Network 70: Safety override - Reset V3245_Nuoc_Bon4
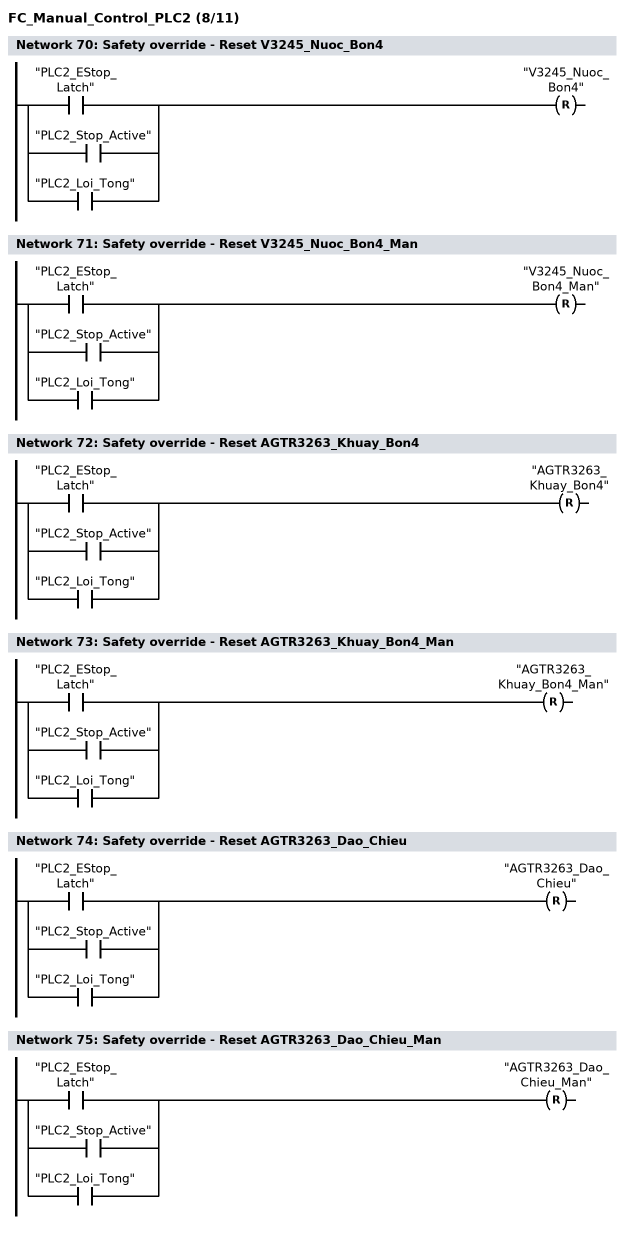
   RUNG wire#powerrail
      Contact( "PLC2_EStop_Latch" )
      wire#w1
      R_Coil( "V3245_Nuoc_Bon4" )
   END_RUNG
   RUNG wire#powerrail
      Contact( "PLC2_Stop_Active" )
   END_RUNG wire#w1
   RUNG wire#powerrail
      Contact( "PLC2_Loi_Tong" )
   END_RUNG wire#w1
   // the same network as SCL:
   IF "PLC2_EStop_Latch" OR "PLC2_Stop_Active" OR "PLC2_Loi_Tong" THEN "V3245_Nuoc_Bon4" := FALSE; END_IF;
END_REGION

REGION Network 71: Safety override - Reset V3245_Nuoc_Bon4_Man
   RUNG wire#powerrail
      Contact( "PLC2_EStop_Latch" )
      wire#w1
      R_Coil( "V3245_Nuoc_Bon4_Man" )
   END_RUNG
   RUNG wire#powerrail
      Contact( "PLC2_Stop_Active" )
   END_RUNG wire#w1
   RUNG wire#powerrail
      Contact( "PLC2_Loi_Tong" )
   END_RUNG wire#w1
   // the same network as SCL:
   IF "PLC2_EStop_Latch" OR "PLC2_Stop_Active" OR "PLC2_Loi_Tong" THEN
       "V3245_Nuoc_Bon4_Man" := FALSE;
   END_IF;
END_REGION

REGION Network 72: Safety override - Reset AGTR3263_Khuay_Bon4
   RUNG wire#powerrail
      Contact( "PLC2_EStop_Latch" )
      wire#w1
      R_Coil( "AGTR3263_Khuay_Bon4" )
   END_RUNG
   RUNG wire#powerrail
      Contact( "PLC2_Stop_Active" )
   END_RUNG wire#w1
   RUNG wire#powerrail
      Contact( "PLC2_Loi_Tong" )
   END_RUNG wire#w1
   // the same network as SCL:
   IF "PLC2_EStop_Latch" OR "PLC2_Stop_Active" OR "PLC2_Loi_Tong" THEN
       "AGTR3263_Khuay_Bon4" := FALSE;
   END_IF;
END_REGION

REGION Network 73: Safety override - Reset AGTR3263_Khuay_Bon4_Man
   RUNG wire#powerrail
      Contact( "PLC2_EStop_Latch" )
      wire#w1
      R_Coil( "AGTR3263_Khuay_Bon4_Man" )
   END_RUNG
   RUNG wire#powerrail
      Contact( "PLC2_Stop_Active" )
   END_RUNG wire#w1
   RUNG wire#powerrail
      Contact( "PLC2_Loi_Tong" )
   END_RUNG wire#w1
   // the same network as SCL:
   IF "PLC2_EStop_Latch" OR "PLC2_Stop_Active" OR "PLC2_Loi_Tong" THEN
       "AGTR3263_Khuay_Bon4_Man" := FALSE;
   END_IF;
END_REGION

REGION Network 74: Safety override - Reset AGTR3263_Dao_Chieu
   RUNG wire#powerrail
      Contact( "PLC2_EStop_Latch" )
      wire#w1
      R_Coil( "AGTR3263_Dao_Chieu" )
   END_RUNG
   RUNG wire#powerrail
      Contact( "PLC2_Stop_Active" )
   END_RUNG wire#w1
   RUNG wire#powerrail
      Contact( "PLC2_Loi_Tong" )
   END_RUNG wire#w1
   // the same network as SCL:
   IF "PLC2_EStop_Latch" OR "PLC2_Stop_Active" OR "PLC2_Loi_Tong" THEN "AGTR3263_Dao_Chieu" := FALSE; END_IF;
END_REGION

REGION Network 75: Safety override - Reset AGTR3263_Dao_Chieu_Man
   RUNG wire#powerrail
      Contact( "PLC2_EStop_Latch" )
      wire#w1
      R_Coil( "AGTR3263_Dao_Chieu_Man" )
   END_RUNG
   RUNG wire#powerrail
      Contact( "PLC2_Stop_Active" )
   END_RUNG wire#w1
   RUNG wire#powerrail
      Contact( "PLC2_Loi_Tong" )
   END_RUNG wire#w1
   // the same network as SCL:
   IF "PLC2_EStop_Latch" OR "PLC2_Stop_Active" OR "PLC2_Loi_Tong" THEN
       "AGTR3263_Dao_Chieu_Man" := FALSE;
   END_IF;
END_REGION

REGION Network 76: Safety override - Reset V3247_Xa_Bon4
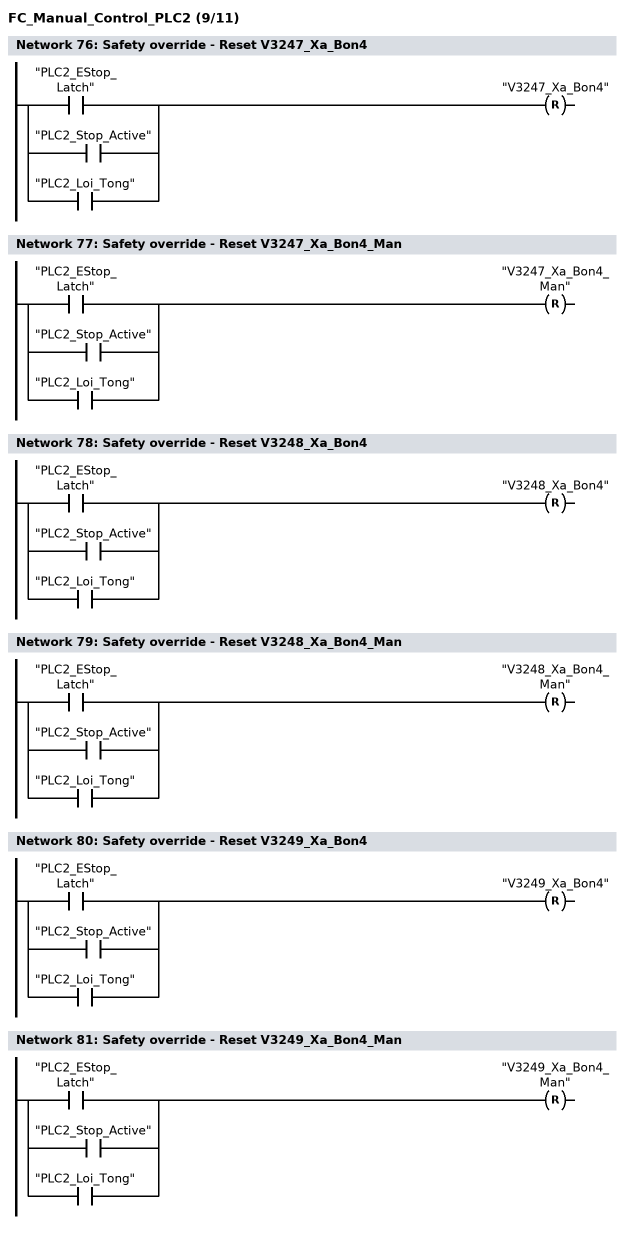
   RUNG wire#powerrail
      Contact( "PLC2_EStop_Latch" )
      wire#w1
      R_Coil( "V3247_Xa_Bon4" )
   END_RUNG
   RUNG wire#powerrail
      Contact( "PLC2_Stop_Active" )
   END_RUNG wire#w1
   RUNG wire#powerrail
      Contact( "PLC2_Loi_Tong" )
   END_RUNG wire#w1
   // the same network as SCL:
   IF "PLC2_EStop_Latch" OR "PLC2_Stop_Active" OR "PLC2_Loi_Tong" THEN "V3247_Xa_Bon4" := FALSE; END_IF;
END_REGION

REGION Network 77: Safety override - Reset V3247_Xa_Bon4_Man
   RUNG wire#powerrail
      Contact( "PLC2_EStop_Latch" )
      wire#w1
      R_Coil( "V3247_Xa_Bon4_Man" )
   END_RUNG
   RUNG wire#powerrail
      Contact( "PLC2_Stop_Active" )
   END_RUNG wire#w1
   RUNG wire#powerrail
      Contact( "PLC2_Loi_Tong" )
   END_RUNG wire#w1
   // the same network as SCL:
   IF "PLC2_EStop_Latch" OR "PLC2_Stop_Active" OR "PLC2_Loi_Tong" THEN "V3247_Xa_Bon4_Man" := FALSE; END_IF;
END_REGION

REGION Network 78: Safety override - Reset V3248_Xa_Bon4
   RUNG wire#powerrail
      Contact( "PLC2_EStop_Latch" )
      wire#w1
      R_Coil( "V3248_Xa_Bon4" )
   END_RUNG
   RUNG wire#powerrail
      Contact( "PLC2_Stop_Active" )
   END_RUNG wire#w1
   RUNG wire#powerrail
      Contact( "PLC2_Loi_Tong" )
   END_RUNG wire#w1
   // the same network as SCL:
   IF "PLC2_EStop_Latch" OR "PLC2_Stop_Active" OR "PLC2_Loi_Tong" THEN "V3248_Xa_Bon4" := FALSE; END_IF;
END_REGION

REGION Network 79: Safety override - Reset V3248_Xa_Bon4_Man
   RUNG wire#powerrail
      Contact( "PLC2_EStop_Latch" )
      wire#w1
      R_Coil( "V3248_Xa_Bon4_Man" )
   END_RUNG
   RUNG wire#powerrail
      Contact( "PLC2_Stop_Active" )
   END_RUNG wire#w1
   RUNG wire#powerrail
      Contact( "PLC2_Loi_Tong" )
   END_RUNG wire#w1
   // the same network as SCL:
   IF "PLC2_EStop_Latch" OR "PLC2_Stop_Active" OR "PLC2_Loi_Tong" THEN "V3248_Xa_Bon4_Man" := FALSE; END_IF;
END_REGION

REGION Network 80: Safety override - Reset V3249_Xa_Bon4
   RUNG wire#powerrail
      Contact( "PLC2_EStop_Latch" )
      wire#w1
      R_Coil( "V3249_Xa_Bon4" )
   END_RUNG
   RUNG wire#powerrail
      Contact( "PLC2_Stop_Active" )
   END_RUNG wire#w1
   RUNG wire#powerrail
      Contact( "PLC2_Loi_Tong" )
   END_RUNG wire#w1
   // the same network as SCL:
   IF "PLC2_EStop_Latch" OR "PLC2_Stop_Active" OR "PLC2_Loi_Tong" THEN "V3249_Xa_Bon4" := FALSE; END_IF;
END_REGION

REGION Network 81: Safety override - Reset V3249_Xa_Bon4_Man
   RUNG wire#powerrail
      Contact( "PLC2_EStop_Latch" )
      wire#w1
      R_Coil( "V3249_Xa_Bon4_Man" )
   END_RUNG
   RUNG wire#powerrail
      Contact( "PLC2_Stop_Active" )
   END_RUNG wire#w1
   RUNG wire#powerrail
      Contact( "PLC2_Loi_Tong" )
   END_RUNG wire#w1
   // the same network as SCL:
   IF "PLC2_EStop_Latch" OR "PLC2_Stop_Active" OR "PLC2_Loi_Tong" THEN "V3249_Xa_Bon4_Man" := FALSE; END_IF;
END_REGION

REGION Network 82: Safety override - Reset Pump3265_Chuyen_Nhanh2
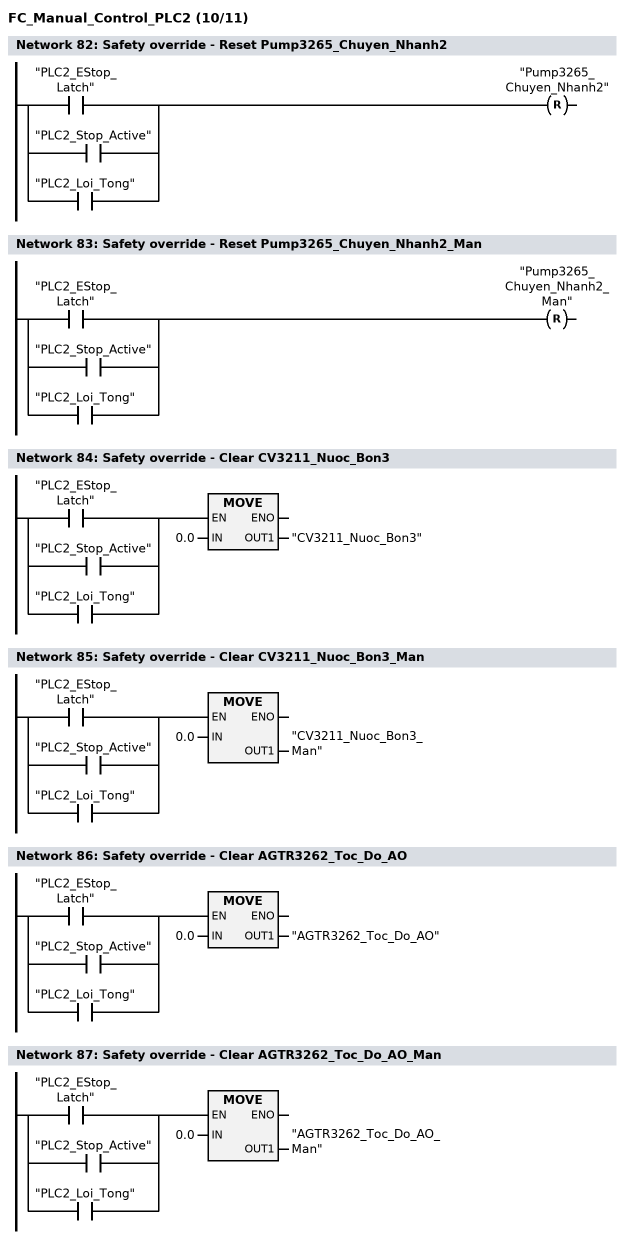
   RUNG wire#powerrail
      Contact( "PLC2_EStop_Latch" )
      wire#w1
      R_Coil( "Pump3265_Chuyen_Nhanh2" )
   END_RUNG
   RUNG wire#powerrail
      Contact( "PLC2_Stop_Active" )
   END_RUNG wire#w1
   RUNG wire#powerrail
      Contact( "PLC2_Loi_Tong" )
   END_RUNG wire#w1
   // the same network as SCL:
   IF "PLC2_EStop_Latch" OR "PLC2_Stop_Active" OR "PLC2_Loi_Tong" THEN
       "Pump3265_Chuyen_Nhanh2" := FALSE;
   END_IF;
END_REGION

REGION Network 83: Safety override - Reset Pump3265_Chuyen_Nhanh2_Man
   RUNG wire#powerrail
      Contact( "PLC2_EStop_Latch" )
      wire#w1
      R_Coil( "Pump3265_Chuyen_Nhanh2_Man" )
   END_RUNG
   RUNG wire#powerrail
      Contact( "PLC2_Stop_Active" )
   END_RUNG wire#w1
   RUNG wire#powerrail
      Contact( "PLC2_Loi_Tong" )
   END_RUNG wire#w1
   // the same network as SCL:
   IF "PLC2_EStop_Latch" OR "PLC2_Stop_Active" OR "PLC2_Loi_Tong" THEN
       "Pump3265_Chuyen_Nhanh2_Man" := FALSE;
   END_IF;
END_REGION

REGION Network 84: Safety override - Clear CV3211_Nuoc_Bon3
   RUNG wire#powerrail
      Contact( "PLC2_EStop_Latch" )
      wire#w1
      { S7_GenerateENO := "TRUE" } Move(in := 0.0, out1 => "CV3211_Nuoc_Bon3")
   END_RUNG
   RUNG wire#powerrail
      Contact( "PLC2_Stop_Active" )
   END_RUNG wire#w1
   RUNG wire#powerrail
      Contact( "PLC2_Loi_Tong" )
   END_RUNG wire#w1
   // the same network as SCL:
   IF "PLC2_EStop_Latch" OR "PLC2_Stop_Active" OR "PLC2_Loi_Tong" THEN "CV3211_Nuoc_Bon3" := 0.0; END_IF;
END_REGION

REGION Network 85: Safety override - Clear CV3211_Nuoc_Bon3_Man
   RUNG wire#powerrail
      Contact( "PLC2_EStop_Latch" )
      wire#w1
      { S7_GenerateENO := "TRUE" } Move(in := 0.0, out1 => "CV3211_Nuoc_Bon3_Man")
   END_RUNG
   RUNG wire#powerrail
      Contact( "PLC2_Stop_Active" )
   END_RUNG wire#w1
   RUNG wire#powerrail
      Contact( "PLC2_Loi_Tong" )
   END_RUNG wire#w1
   // the same network as SCL:
   IF "PLC2_EStop_Latch" OR "PLC2_Stop_Active" OR "PLC2_Loi_Tong" THEN "CV3211_Nuoc_Bon3_Man" := 0.0; END_IF;
END_REGION

REGION Network 86: Safety override - Clear AGTR3262_Toc_Do_AO
   RUNG wire#powerrail
      Contact( "PLC2_EStop_Latch" )
      wire#w1
      { S7_GenerateENO := "TRUE" } Move(in := 0.0, out1 => "AGTR3262_Toc_Do_AO")
   END_RUNG
   RUNG wire#powerrail
      Contact( "PLC2_Stop_Active" )
   END_RUNG wire#w1
   RUNG wire#powerrail
      Contact( "PLC2_Loi_Tong" )
   END_RUNG wire#w1
   // the same network as SCL:
   IF "PLC2_EStop_Latch" OR "PLC2_Stop_Active" OR "PLC2_Loi_Tong" THEN "AGTR3262_Toc_Do_AO" := 0.0; END_IF;
END_REGION

REGION Network 87: Safety override - Clear AGTR3262_Toc_Do_AO_Man
   RUNG wire#powerrail
      Contact( "PLC2_EStop_Latch" )
      wire#w1
      { S7_GenerateENO := "TRUE" } Move(in := 0.0, out1 => "AGTR3262_Toc_Do_AO_Man")
   END_RUNG
   RUNG wire#powerrail
      Contact( "PLC2_Stop_Active" )
   END_RUNG wire#w1
   RUNG wire#powerrail
      Contact( "PLC2_Loi_Tong" )
   END_RUNG wire#w1
   // the same network as SCL:
   IF "PLC2_EStop_Latch" OR "PLC2_Stop_Active" OR "PLC2_Loi_Tong" THEN
       "AGTR3262_Toc_Do_AO_Man" := 0.0;
   END_IF;
END_REGION

REGION Network 88: Safety override - Clear CV3216_Hoi_Bon4
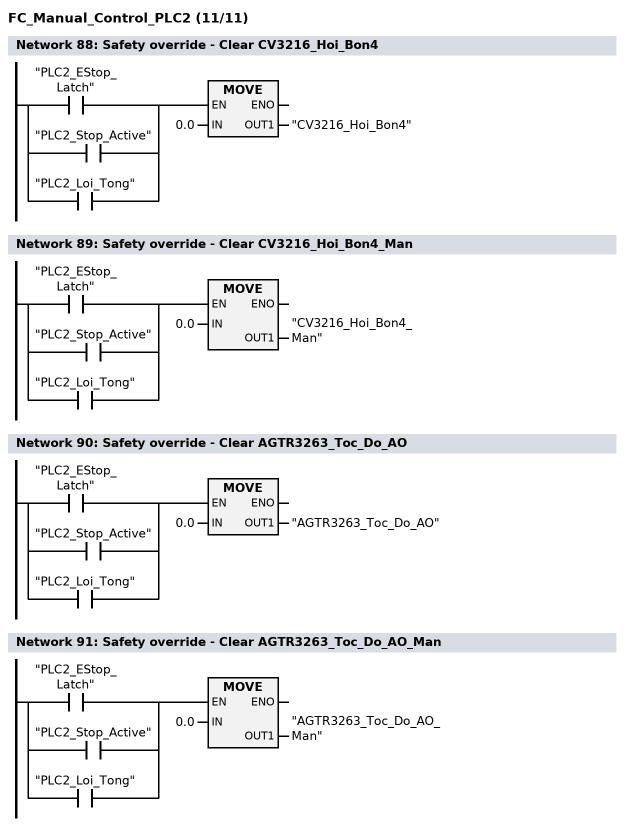
   RUNG wire#powerrail
      Contact( "PLC2_EStop_Latch" )
      wire#w1
      { S7_GenerateENO := "TRUE" } Move(in := 0.0, out1 => "CV3216_Hoi_Bon4")
   END_RUNG
   RUNG wire#powerrail
      Contact( "PLC2_Stop_Active" )
   END_RUNG wire#w1
   RUNG wire#powerrail
      Contact( "PLC2_Loi_Tong" )
   END_RUNG wire#w1
   // the same network as SCL:
   IF "PLC2_EStop_Latch" OR "PLC2_Stop_Active" OR "PLC2_Loi_Tong" THEN "CV3216_Hoi_Bon4" := 0.0; END_IF;
END_REGION

REGION Network 89: Safety override - Clear CV3216_Hoi_Bon4_Man
   RUNG wire#powerrail
      Contact( "PLC2_EStop_Latch" )
      wire#w1
      { S7_GenerateENO := "TRUE" } Move(in := 0.0, out1 => "CV3216_Hoi_Bon4_Man")
   END_RUNG
   RUNG wire#powerrail
      Contact( "PLC2_Stop_Active" )
   END_RUNG wire#w1
   RUNG wire#powerrail
      Contact( "PLC2_Loi_Tong" )
   END_RUNG wire#w1
   // the same network as SCL:
   IF "PLC2_EStop_Latch" OR "PLC2_Stop_Active" OR "PLC2_Loi_Tong" THEN "CV3216_Hoi_Bon4_Man" := 0.0; END_IF;
END_REGION

REGION Network 90: Safety override - Clear AGTR3263_Toc_Do_AO
   RUNG wire#powerrail
      Contact( "PLC2_EStop_Latch" )
      wire#w1
      { S7_GenerateENO := "TRUE" } Move(in := 0.0, out1 => "AGTR3263_Toc_Do_AO")
   END_RUNG
   RUNG wire#powerrail
      Contact( "PLC2_Stop_Active" )
   END_RUNG wire#w1
   RUNG wire#powerrail
      Contact( "PLC2_Loi_Tong" )
   END_RUNG wire#w1
   // the same network as SCL:
   IF "PLC2_EStop_Latch" OR "PLC2_Stop_Active" OR "PLC2_Loi_Tong" THEN "AGTR3263_Toc_Do_AO" := 0.0; END_IF;
END_REGION

REGION Network 91: Safety override - Clear AGTR3263_Toc_Do_AO_Man
   RUNG wire#powerrail
      Contact( "PLC2_EStop_Latch" )
      wire#w1
      { S7_GenerateENO := "TRUE" } Move(in := 0.0, out1 => "AGTR3263_Toc_Do_AO_Man")
   END_RUNG
   RUNG wire#powerrail
      Contact( "PLC2_Stop_Active" )
   END_RUNG wire#w1
   RUNG wire#powerrail
      Contact( "PLC2_Loi_Tong" )
   END_RUNG wire#w1
   // the same network as SCL:
   IF "PLC2_EStop_Latch" OR "PLC2_Stop_Active" OR "PLC2_Loi_Tong" THEN
       "AGTR3263_Toc_Do_AO_Man" := 0.0;
   END_IF;
END_REGION
END_FUNCTION
